TYPE ST_CtrlInClosedPalletCheck :
STRUCT
	ExternalTrigger : BOOL;
	ExternalNumberOfFingersOk : INT;
	
END_STRUCT
END_TYPE

(* stored: Version 1.1.0.1, ProductVersion 3.1.4024.9
   DUT ST_CtrlInClosedPalletCheck: Id {90c37ad0-83c6-49c9-b6b7-691dcfc51515} *)
